FUNCTION_BLOCK FB_Conveyor_Sim IMPLEMENTS I_Conveyor
VAR_INPUT
END_VAR
VAR_OUTPUT
END_VAR
VAR
	bRunConveyor : BOOL;
	bIsRun		 : BOOL;
END_VAR

IF bRunConveyor THEN
	bIsRun := TRUE;
ELSE
	bIsRun := FALSE;
END_IF

PROPERTY IsRun : BOOL
GET
IsRun := bIsRun;
END_GET
END_PROPERTY

METHOD Start : BOOL
VAR_INPUT
END_VAR
bRunConveyor := TRUE;
END_METHOD

METHOD Stop : BOOL
VAR_INPUT
END_VAR
bRunConveyor := FALSE;
END_METHOD

END_FUNCTION_BLOCK

(* stored: Version 1.1.0.1, ProductVersion 3.1.4024.12
   POU FB_Conveyor_Sim: Id {5b50461e-6d34-4e99-b7e5-480daff7770c}, SpecialFunc None
   Property IsRun: Id {f56fba4c-cef9-4421-a910-cfdcc706e4f6}
   Get Get: Id {2fb5369b-d6b4-41d9-9fb0-c05eb2f42731}
   Method Start: Id {64b8eb14-af7d-4e19-ac48-8ba72824c50a}
   Method Stop: Id {d8f0f0ad-9e0e-4ea2-a736-3e1fee03f61d} *)
